Omron CX-Programmer project NewProject (CX-Programmer 9.81)

# PLC Sessao_01_04_2026_Exercicio: CP1L M

## Global symbols (name address type ; comment)
0.00 BOOL  ; Botao Start
0.01 BOOL  ; Temporizador 1
0.02 BOOL  ; Flag do Temporizador 1
0.03 BOOL  ; Botao Stop
0.04 BOOL  ; Botao Start
0.05 BOOL  ; Botao Start 1
0.06 BOOL  ; Botao de Emergencia 2
0.07 BOOL  ; Botao Stop 1
0.08 BOOL  ; Flag do Temporizador 1
0.09 BOOL  ; Botao de Start Esquerdo
0.10 BOOL  ; Botao de Start Direito
0.11 BOOL  ; Temporizador
100 CHANNEL  ; Temporizador
100.00 BOOL  ; Contactor
100.01 BOOL  ; Lampada 2
100.02 BOOL  ; Lampada 3
100.03 BOOL  ; Lampada 4
100.04 BOOL  ; Bobina do Rele
100.05 BOOL  ; Bobina do Motor 1
100.06 BOOL  ; Bobina do Motor 2
100.07 BOOL  ; Temporizador
500 CHANNEL  ; Temporizador 1
T0001 BOOL  ; Flag do Temporizador 1

## Program NewProgram1 (cyclic task 0)
Local symbols
Flag_T1 T0001 BOOL  ; Flag do temporizador
T 1 NUMBER  ; Temporizador
Tempo_T #5 NUMBER  ; Tempo do Temporizador
V1 100.01 BOOL  ; Velocidade 1
V2 100.02 BOOL  ; Velocidade 2
V3 100.03 BOOL  ; Velocidade 3
b1 0.00 BOOL  ; Botao 1
b2 0.01 BOOL  ; Botao 2
b3 0.02 BOOL  ; Botao 3
etapa_0 2.00 BOOL  ; Etapa 0 do Grafcet
etapa_1 2.01 BOOL  ; Etapa 1 do Grafcet

### Section Exercicio

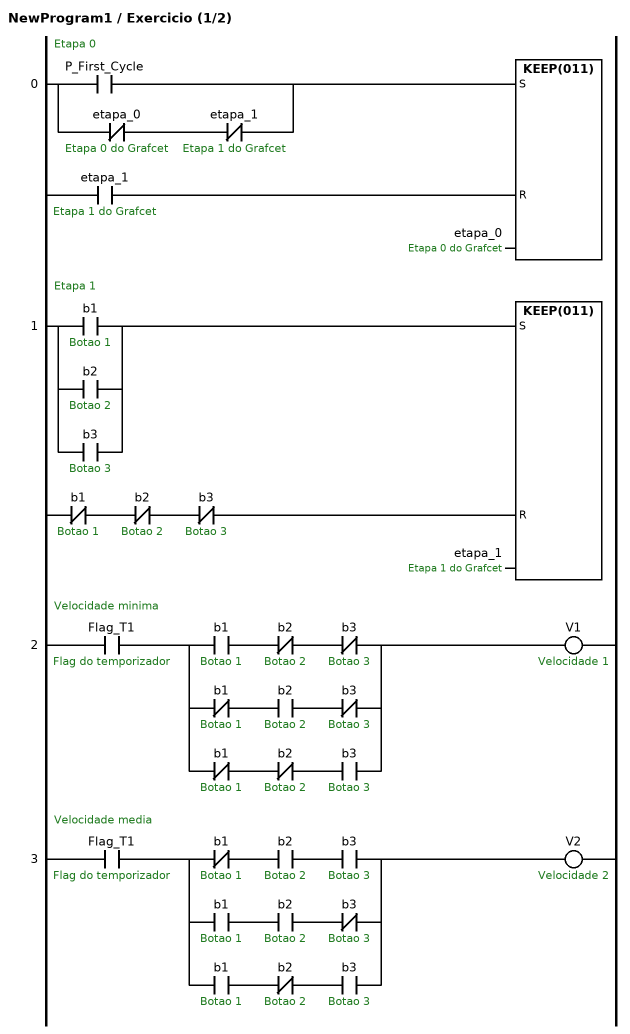
; rung 0: Etapa 0
LD P_First_Cycle
LDNOT etapa_0  ; Etapa 0 do Grafcet
ANDNOT etapa_1  ; Etapa 1 do Grafcet
ORLD
LD etapa_1  ; Etapa 1 do Grafcet
KEEP(011) etapa_0  ; Etapa 0 do Grafcet
; rung 1: Etapa 1
LD b1  ; Botao 1
OR b2  ; Botao 2
OR b3  ; Botao 3
LDNOT b1  ; Botao 1
ANDNOT b2  ; Botao 2
ANDNOT b3  ; Botao 3
KEEP(011) etapa_1  ; Etapa 1 do Grafcet
; rung 2: Velocidade minima
LD Flag_T1  ; Flag do temporizador
LD b1  ; Botao 1
ANDNOT b2  ; Botao 2
ANDNOT b3  ; Botao 3
LDNOT b1  ; Botao 1
AND b2  ; Botao 2
ANDNOT b3  ; Botao 3
ORLD
LDNOT b1  ; Botao 1
ANDNOT b2  ; Botao 2
AND b3  ; Botao 3
ORLD
ANDLD
OUT V1  ; Velocidade 1
; rung 3: Velocidade media
LD Flag_T1  ; Flag do temporizador
LDNOT b1  ; Botao 1
AND b2  ; Botao 2
AND b3  ; Botao 3
LD b1  ; Botao 1
AND b2  ; Botao 2
ANDNOT b3  ; Botao 3
ORLD
LD b1  ; Botao 1
ANDNOT b2  ; Botao 2
AND b3  ; Botao 3
ORLD
ANDLD
OUT V2  ; Velocidade 2

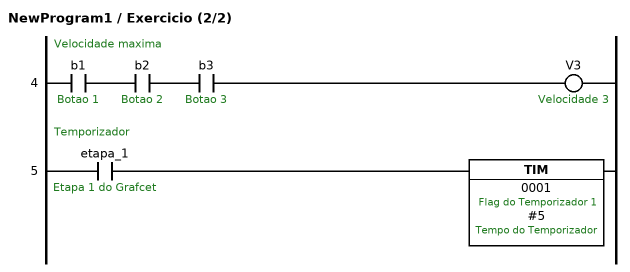
; rung 4: Velocidade maxima
LD b1  ; Botao 1
AND b2  ; Botao 2
AND b3  ; Botao 3
OUT V3  ; Velocidade 3
; rung 5: Temporizador
LD etapa_1  ; Etapa 1 do Grafcet
TIM 0001 #5  ; Tempo do Temporizador, Flag do Temporizador 1

### Section END
; rung 0
END(001)